Universal Robots PolyScope program: NIST connector.urp

Program NIST connector (installation=default directory=/programs createdIn=5.9.1.1031110 lastSavedIn=5.9.1.1031110 robotSerialNumber=20195501059)
Calibrated DH parameters: a=[0.000146, -0.418764, -0.053981, 0.000058, -0.000023, 0]; d=[0.162545, 37.319448, -206.067439, 168.881546, 0.09955, 0.099464]; alpha=[1.57004, -0.001979, 0.002304, 1.570607, -1.57066, 0]; deltaTheta=[0, -0.174616, -1.258233, 1.432844, -0.000001, 0]
BeforeStart
  URCap Gripper Activate (Robotiq_Grippers, Robotiq Inc.) dataModel(ResetAndActivateKey=false)
  start_p := get_actual_tcp_pose()
  MoveJ speed 60 deg/s, acceleration 80 deg/s^2 (useActiveTCP=true) feature=Base
    Waypoint Waypoint (Variable): variable=start_p
Robot Program (runOnlyOnce=true)
  MoveL speed 250 mm/s, acceleration 1200 mm/s^2 (useActiveTCP=true) feature=Base
    Waypoint home_p: TCP in base x=380.085 y=-194.418 z=124.365 mm, rx=-2.2204 ry=-2.2225 rz=-0.0001 rad; joints [134.67, -95.2, 123.81, -118.602, 270.068, 134.631] deg; TCP offset x=0 y=0 z=174 mm, rx=0 ry=0 rz=0 rad
  Call pick_from_table
  Call insert
  Call remove
  Call return_to_table
SubProgram  [hidden by the author, left out]
SubProgram  [hidden by the author, left out]
SubProgram  [hidden by the author, left out]
SubProgram  [hidden by the author, left out]
SubProgram pick_from_table [hidden by the author, left out]
SubProgram insert [hidden by the author, left out]
SubProgram remove [hidden by the author, left out]
SubProgram return_to_table [hidden by the author, left out]
